TYPE ST_Event :
STRUCT
	

END_STRUCT
END_TYPE

(* stored: Version 1.1.0.1, ProductVersion 3.1.4024.16
   DUT ST_Event: Id {856ad31a-a910-410b-9dc2-64c2badbea97} *)
